// SIMATIC S7-200 project (STEP 7-Micro/WIN), CPU 224 REL 02.01

ORGANIZATION_BLOCK 主程序:OB1
TITLE=程序注释
BEGIN
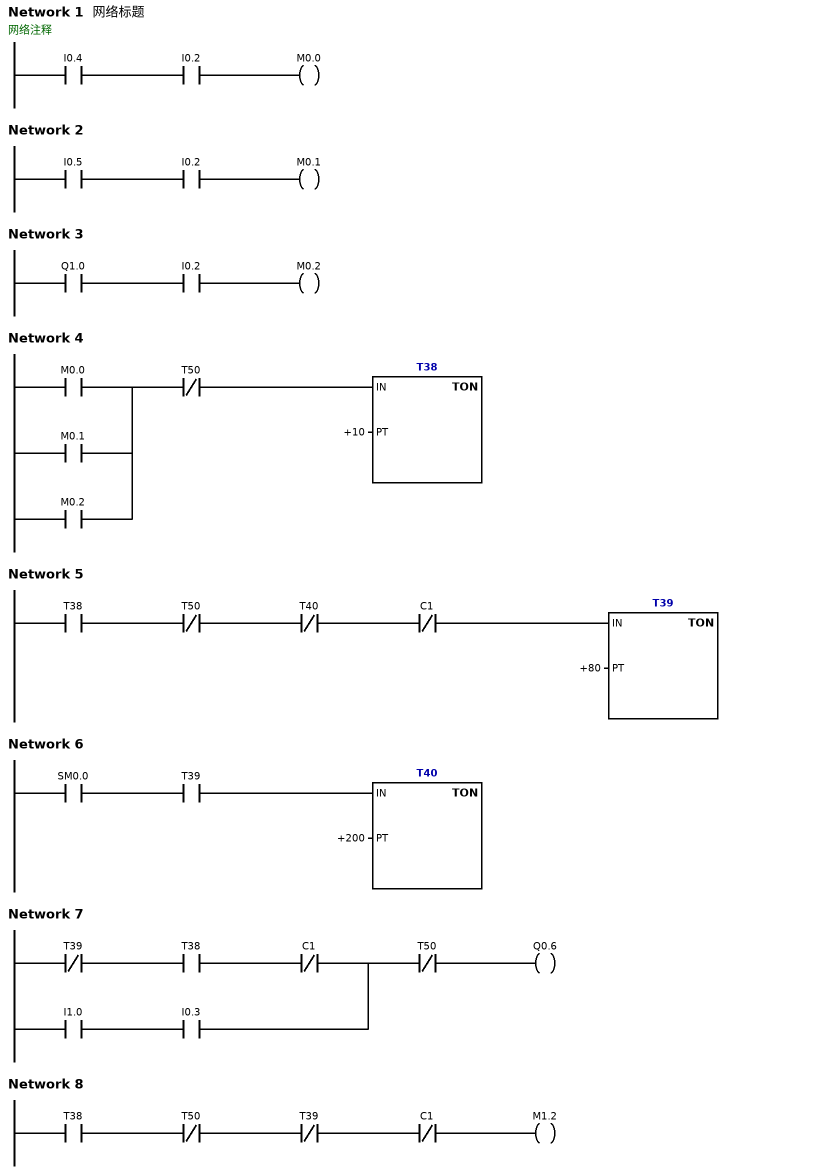
Network 1 // 网络标题
// 网络注释
LD     I0.4
A      I0.2
=      M0.0
Network 2
LD     I0.5
A      I0.2
=      M0.1
Network 3
LD     Q1.0
A      I0.2
=      M0.2
Network 4
LD     M0.0
O      M0.1
O      M0.2
AN     T50
TON    T38, +10
Network 5
LD     T38
AN     T50
AN     T40
AN     C1
TON    T39, +80
Network 6
LD     SM0.0
A      T39
TON    T40, +200
Network 7
LDN    T39
A      T38
AN     C1
LD     I1.0
A      I0.3
OLD
AN     T50
=      Q0.6
Network 8
LD     T38
AN     T50
AN     T39
AN     C1
=      M1.2
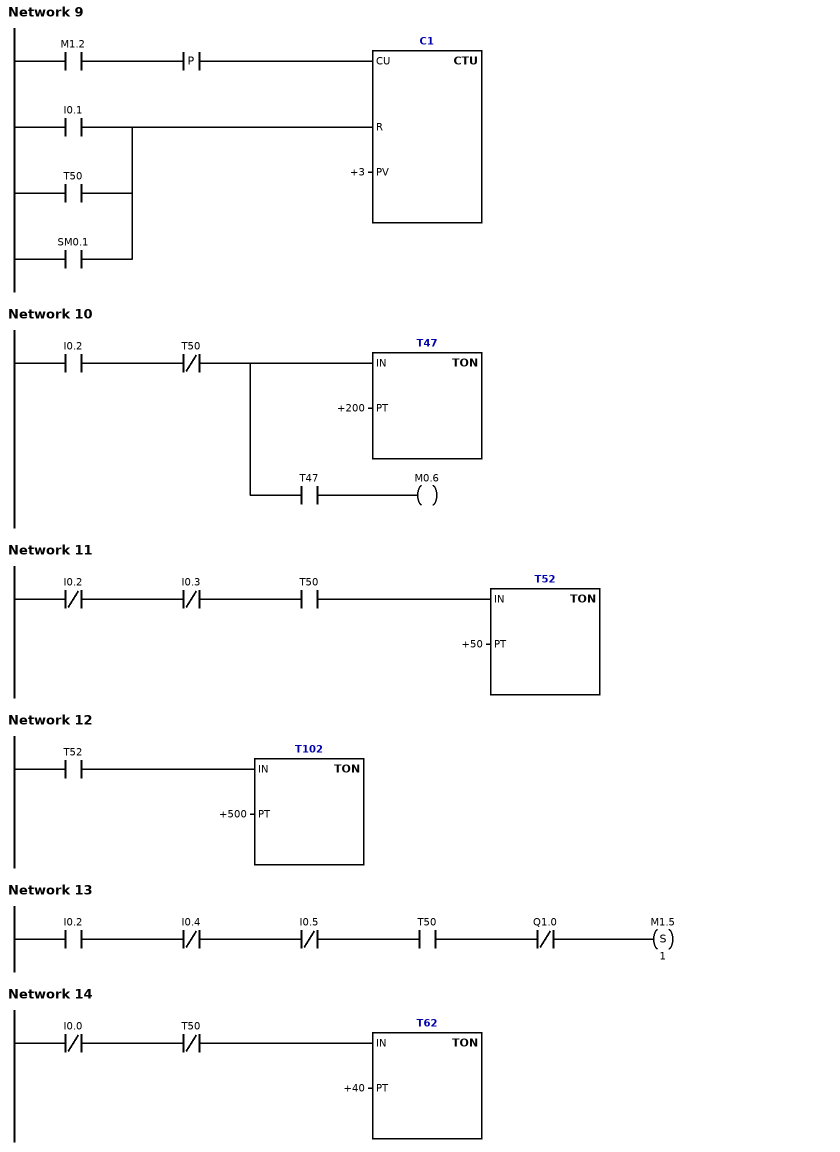
Network 9
LD     M1.2
EU
LD     I0.1
O      T50
O      SM0.1
CTU    C1, +3
Network 10
LD     I0.2
AN     T50
TON    T47, +200
A      T47
=      M0.6
Network 11
LDN    I0.2
AN     I0.3
A      T50
TON    T52, +50
Network 12
LD     T52
TON    T102, +500
Network 13
LD     I0.2
AN     I0.4
AN     I0.5
A      T50
AN     Q1.0
S      M1.5, 1
Network 14
LDN    I0.0
AN     T50
TON    T62, +40
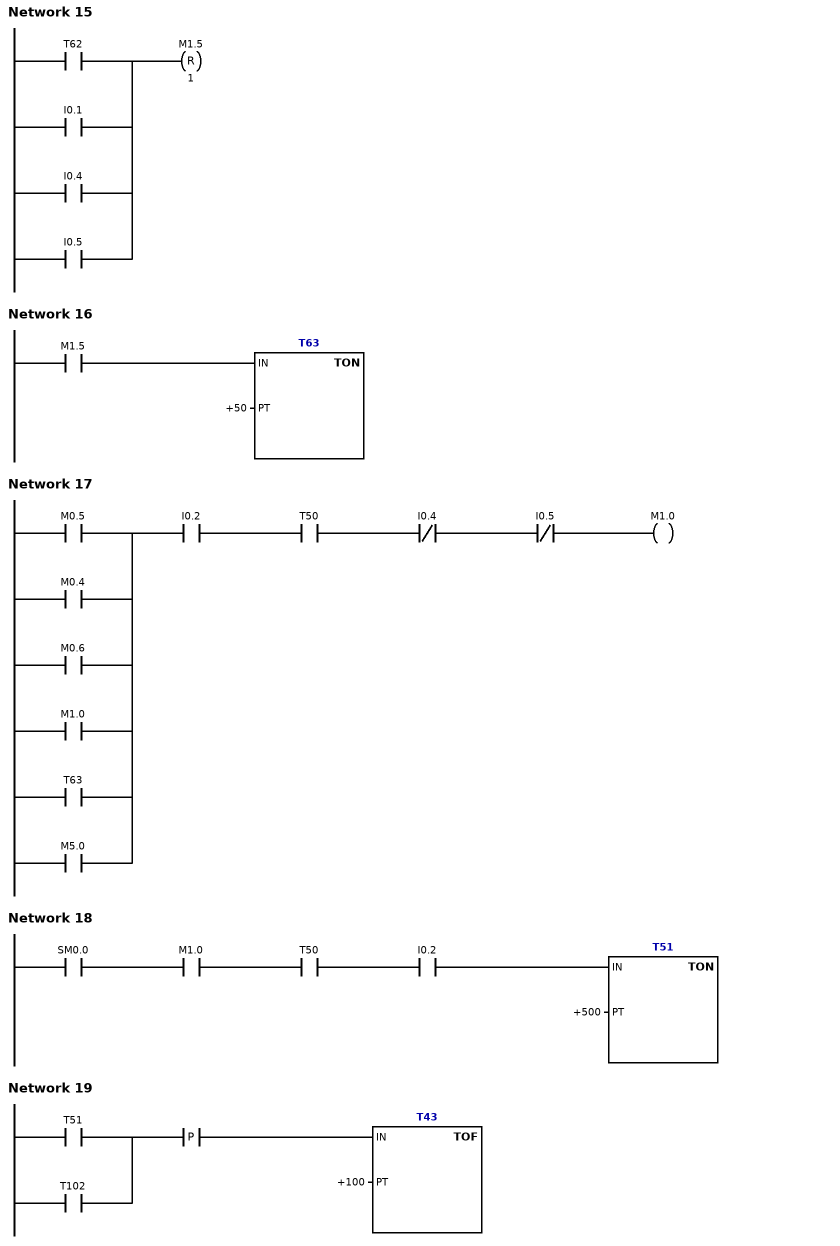
Network 15
LD     T62
O      I0.1
O      I0.4
O      I0.5
R      M1.5, 1
Network 16
LD     M1.5
TON    T63, +50
Network 17
LD     M0.5
O      M0.4
O      M0.6
O      M1.0
O      T63
O      M5.0
A      I0.2
A      T50
AN     I0.4
AN     I0.5
=      M1.0
Network 18
LD     SM0.0
A      M1.0
A      T50
A      I0.2
TON    T51, +500
Network 19
LD     T51
O      T102
EU
TOF    T43, +100
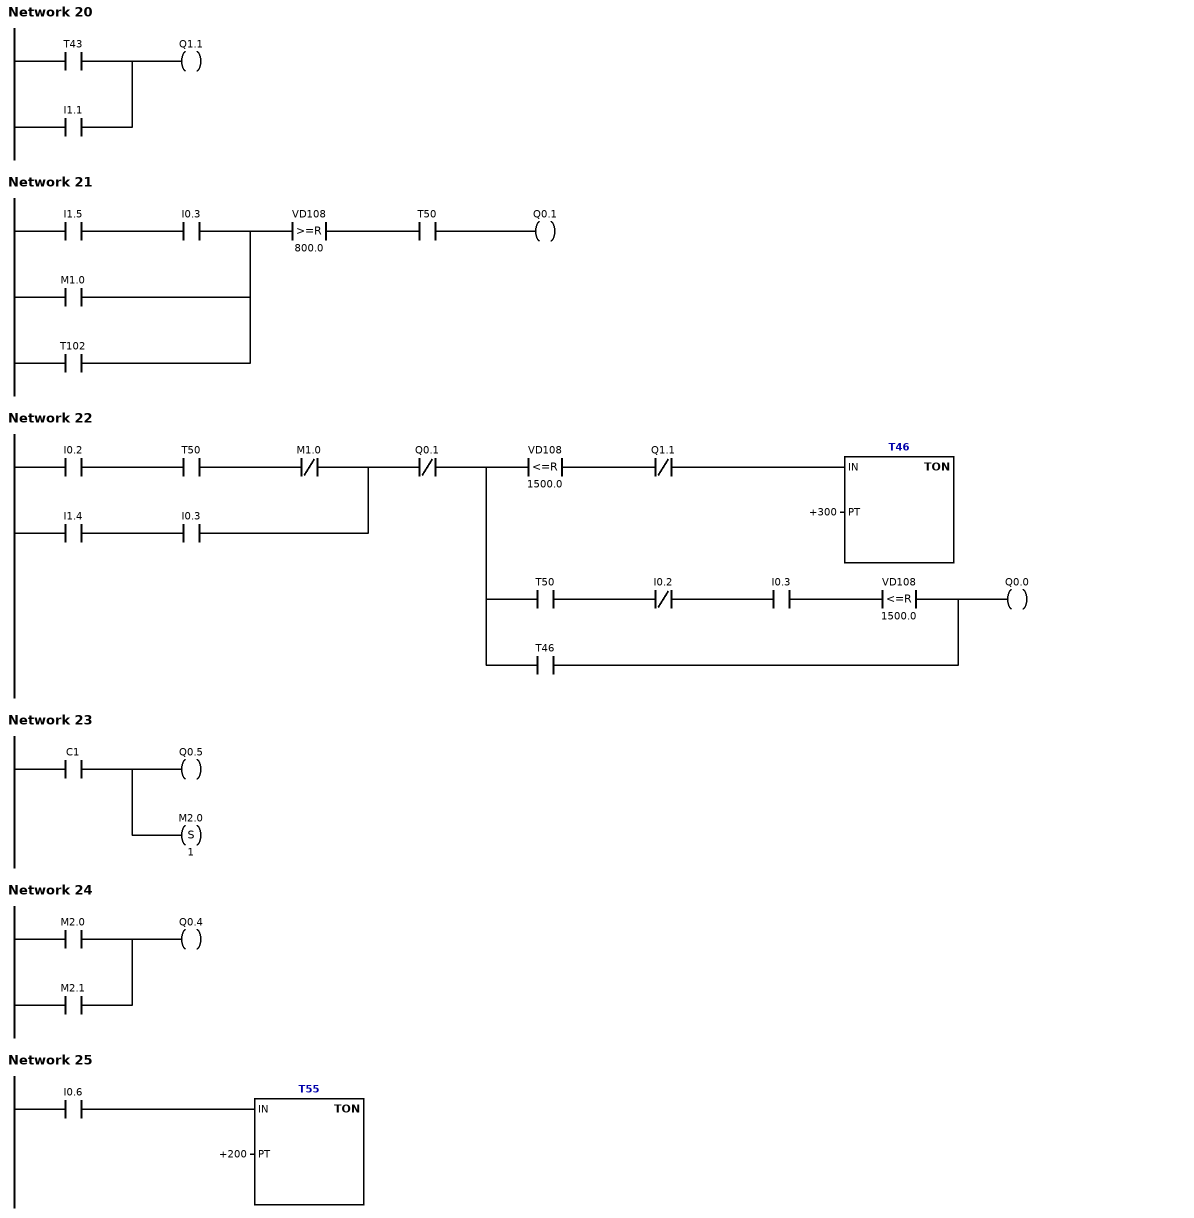
Network 20
LD     T43
O      I1.1
=      Q1.1
Network 21
LD     I1.5
A      I0.3
O      M1.0
O      T102
AR>=   VD108, 800.0
A      T50
=      Q0.1
Network 22
LD     I0.2
A      T50
AN     M1.0
LD     I1.4
A      I0.3
OLD
AN     Q0.1
LPS
AR<=   VD108, 1500.0
AN     Q1.1
TON    T46, +300
LPP
LD     T50
AN     I0.2
A      I0.3
AR<=   VD108, 1500.0
O      T46
ALD
=      Q0.0
Network 23
LD     C1
=      Q0.5
S      M2.0, 1
Network 24
LD     M2.0
O      M2.1
=      Q0.4
Network 25
LD     I0.6
TON    T55, +200
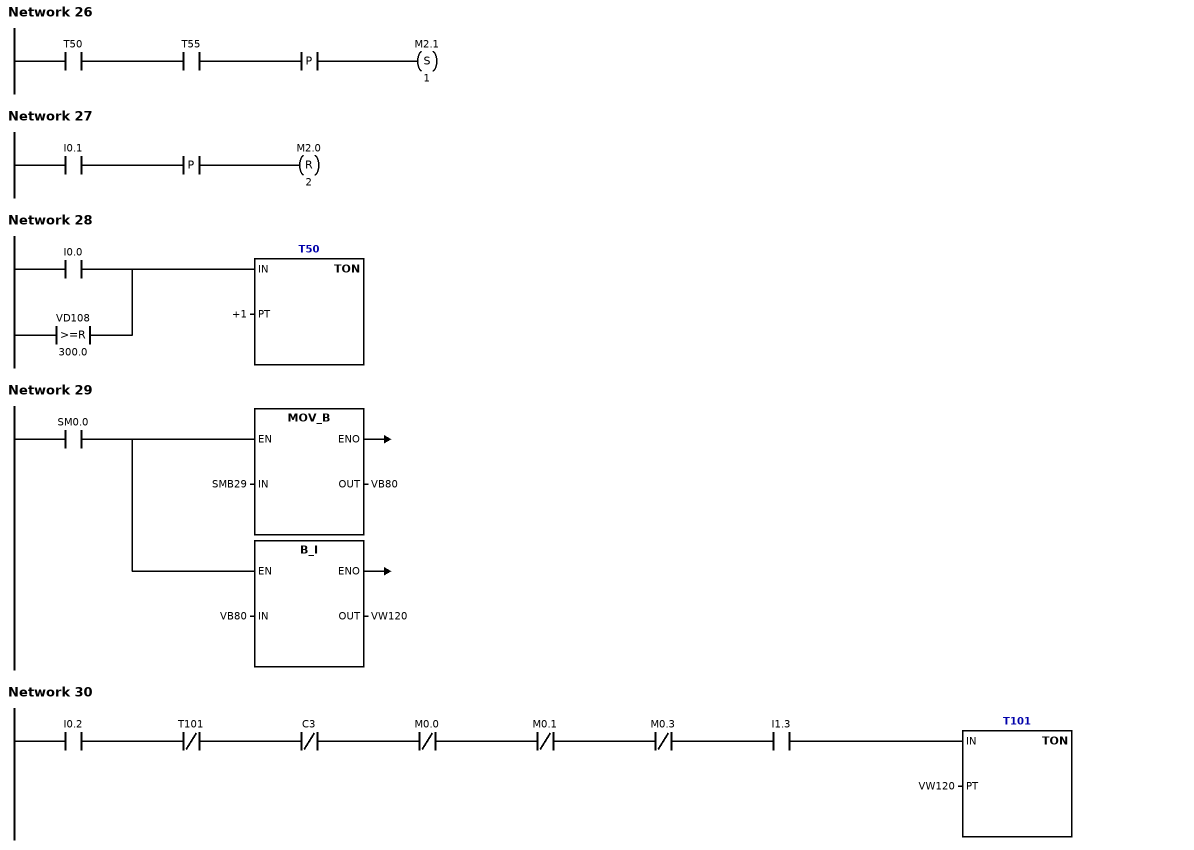
Network 26
LD     T50
A      T55
EU
S      M2.1, 1
Network 27
LD     I0.1
EU
R      M2.0, 2
Network 28
LD     I0.0
OR>=   VD108, 300.0
TON    T50, +1
Network 29
LD     SM0.0
MOVB   SMB29, VB80
BTI    VB80, VW120
Network 30
LD     I0.2
AN     T101
AN     C3
AN     M0.0
AN     M0.1
AN     M0.3
A      I1.3
TON    T101, VW120
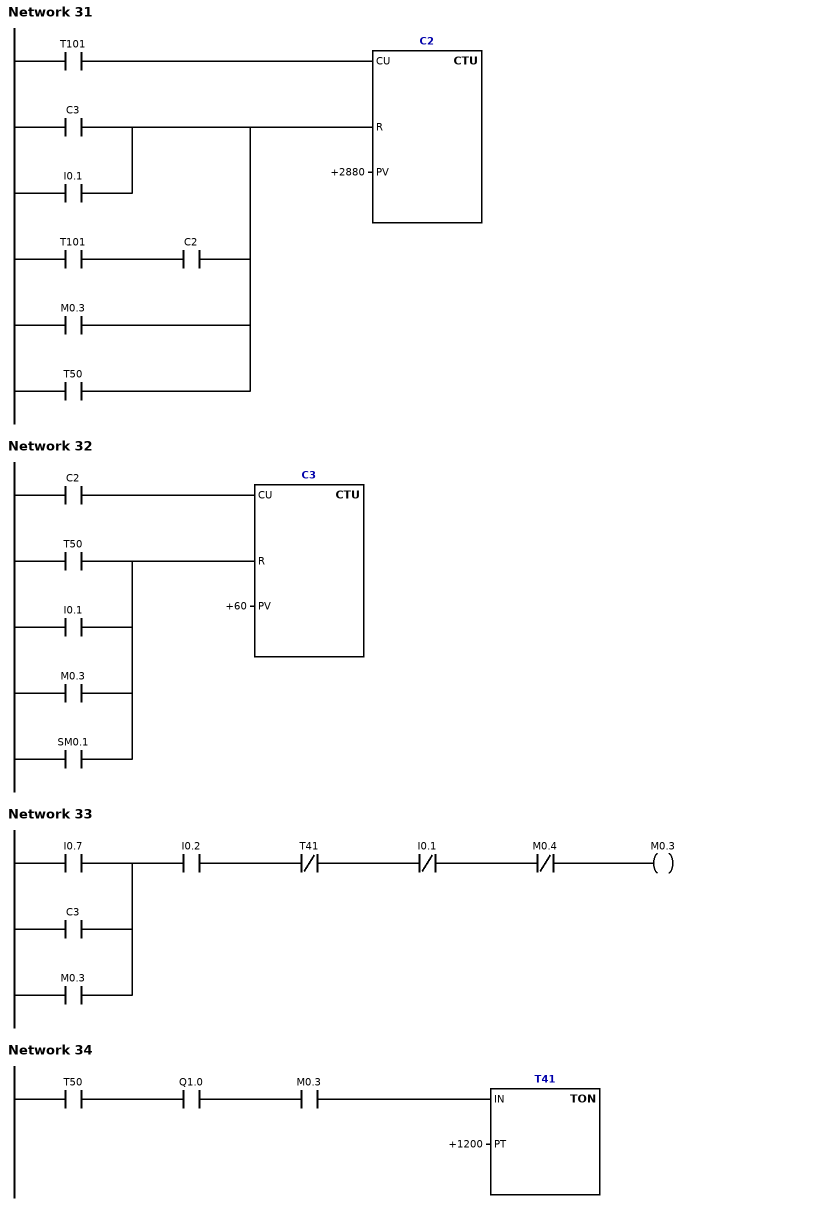
Network 31
LD     T101
LD     C3
O      I0.1
LD     T101
A      C2
OLD
O      M0.3
O      T50
CTU    C2, +2880
Network 32
LD     C2
LD     T50
O      I0.1
O      M0.3
O      SM0.1
CTU    C3, +60
Network 33
LD     I0.7
O      C3
O      M0.3
A      I0.2
AN     T41
AN     I0.1
AN     M0.4
=      M0.3
Network 34
LD     T50
A      Q1.0
A      M0.3
TON    T41, +1200
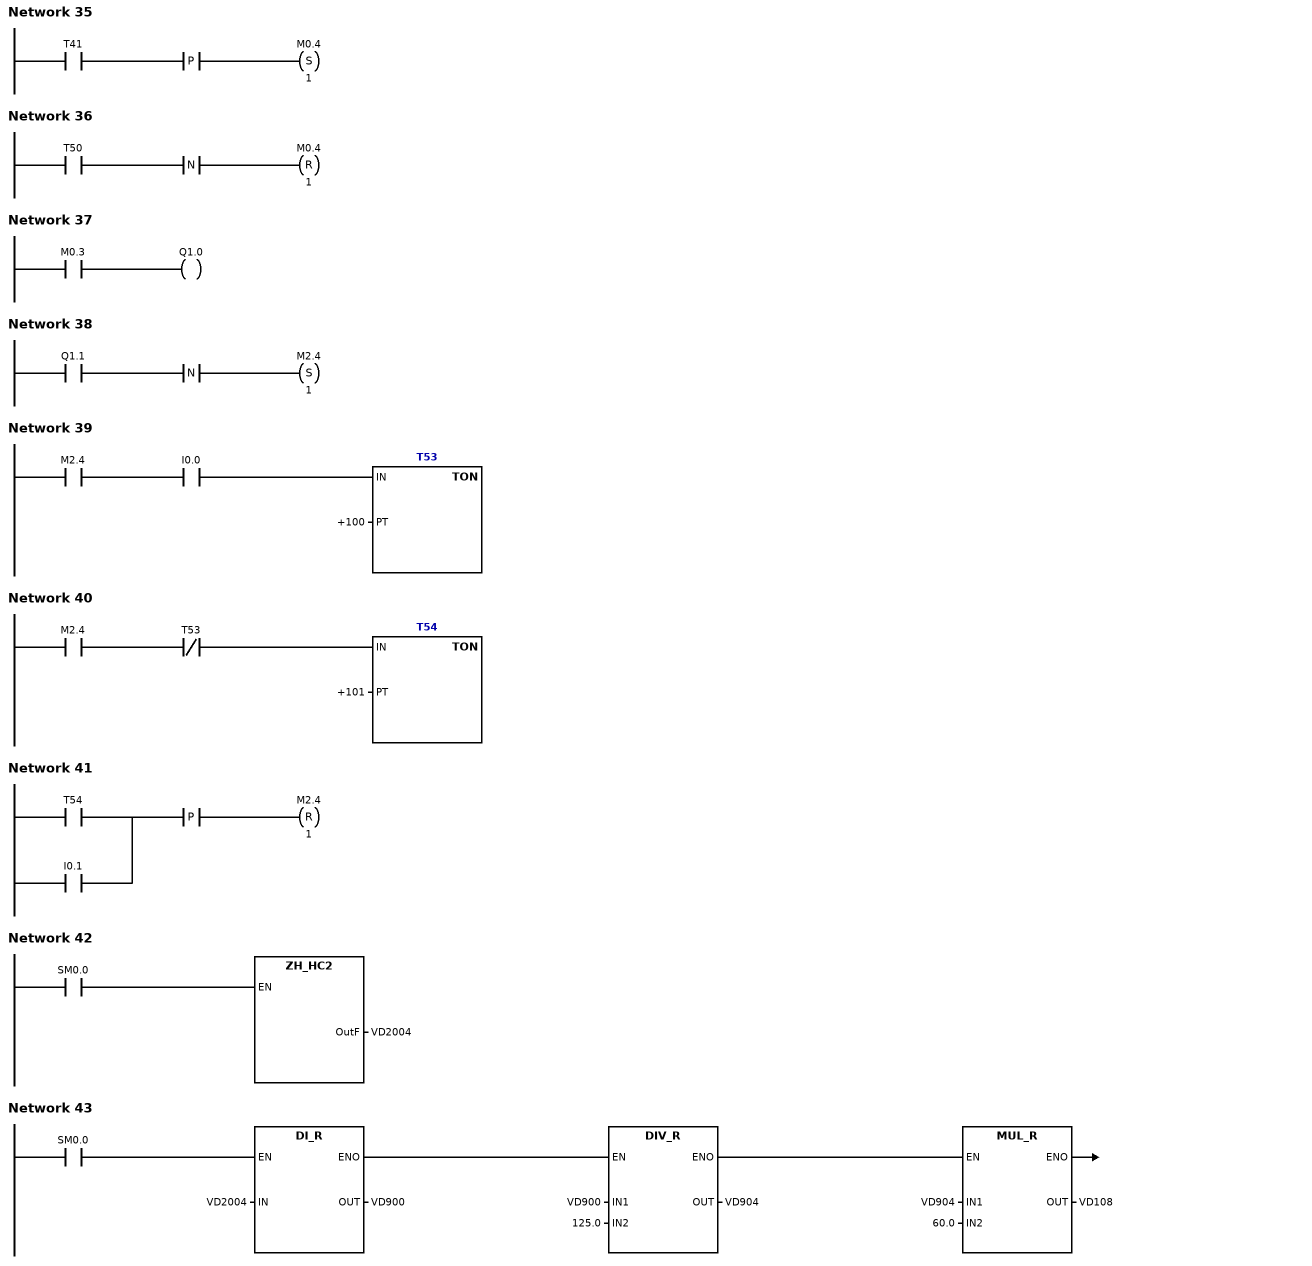
Network 35
LD     T41
EU
S      M0.4, 1
Network 36
LD     T50
ED
R      M0.4, 1
Network 37
LD     M0.3
=      Q1.0
Network 38
LD     Q1.1
ED
S      M2.4, 1
Network 39
LD     M2.4
A      I0.0
TON    T53, +100
Network 40
LD     M2.4
AN     T53
TON    T54, +101
Network 41
LD     T54
O      I0.1
EU
R      M2.4, 1
Network 42
LD     SM0.0
CALL   ZH_HC2:SBR1, VD2004
Network 43
LD     SM0.0
DTR    VD2004, VD900
AENO
MOVR   VD900, VD904
AENO
/R     125.0, VD904
AENO
MOVR   VD904, VD108
*R     60.0, VD108
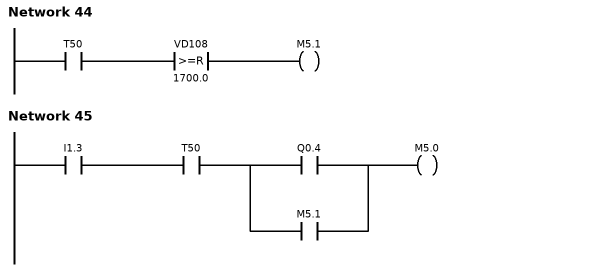
Network 44
LD     T50
AR>=   VD108, 1700.0
=      M5.1
Network 45
LD     I1.3
A      T50
LD     Q0.4
O      M5.1
ALD
=      M5.0
END_ORGANIZATION_BLOCK

// SBR1: protected block, not included
